FUNCTION_BLOCK SUBL_119_BOTTOM_AND_SIDE_ROUGH_MILLING-SLOT-SIMPLE (* 119-variable local group subscriber *)
  (* Standard: 61499-2 *)
  (* Version 1.0, 10-05-12, GASR, Universidade do Estado de Santa Catarina *)
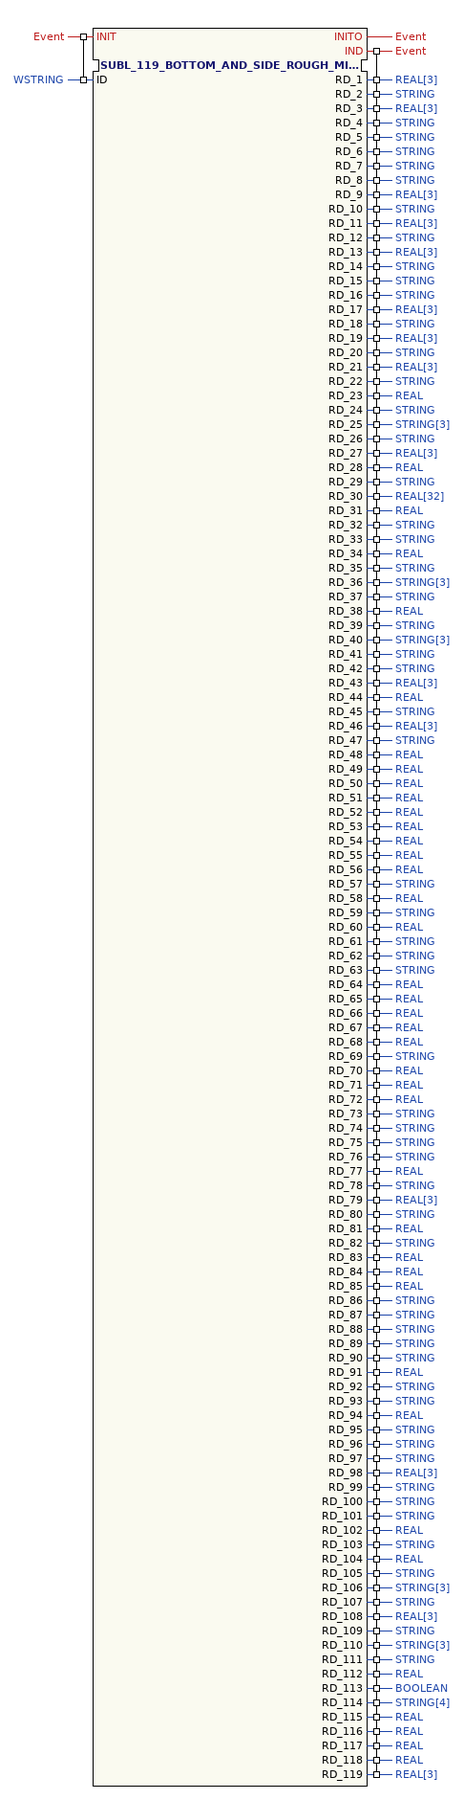
  EVENT_INPUT
    INIT WITH ID; (* Service Initialization *)
  END_EVENT
  EVENT_OUTPUT
    INITO; (* Initialization Confirm *)
    IND WITH RD_1, RD_2, RD_3, RD_4, RD_5, RD_6, RD_7, RD_8, RD_9, RD_10, RD_11, RD_12, RD_13, RD_14, RD_15, RD_16, RD_17, RD_18, RD_19, RD_20, RD_21, RD_22, RD_23, RD_24, RD_25, RD_26, RD_27, RD_28, RD_29, RD_30, RD_31, RD_32, RD_33, RD_34, RD_35, RD_36, RD_37, RD_38, RD_39, RD_40, RD_41, RD_42, RD_43, RD_44, RD_45, RD_46, RD_47, RD_48, RD_49, RD_50, RD_51, RD_52, RD_53, RD_54, RD_55, RD_56, RD_57, RD_58, RD_59, RD_60, RD_61, RD_62, RD_63, RD_64, RD_65, RD_66, RD_67, RD_68, RD_69, RD_70, RD_71, RD_72, RD_73, RD_74, RD_75, RD_76, RD_77, RD_78, RD_79, RD_80, RD_81, RD_82, RD_83, RD_84, RD_85, RD_86, RD_87, RD_88, RD_89, RD_90, RD_91, RD_92, RD_93, RD_94, RD_95, RD_96, RD_97, RD_98, RD_99, RD_100, RD_101, RD_102, RD_103, RD_104, RD_105, RD_106, RD_107, RD_108, RD_109, RD_110, RD_111, RD_112, RD_113, RD_114, RD_115, RD_116, RD_117, RD_118, RD_119; (* Service Indication *)
  END_EVENT
  VAR_INPUT
    ID : WSTRING; (* Default id is the FB instance name *)
  END_VAR
  VAR_OUTPUT
    RD_1 : ARRAY [0..2] OF REAL; (* pos *)
    RD_2 : STRING; (* current_tool *)
    RD_3 : ARRAY [0..2] OF REAL; (* setup.Its_secplane.position.location.coordinates *)
    RD_4 : STRING; (* slot.its_id *)
    RD_5 : STRING; (* its_workpiece.its_id *)
    RD_6 : STRING; (* its_operations.its_id LIST - the list is concatenated in one string *)
    RD_7 : STRING; (* feature_placement.name *)
    RD_8 : STRING; (* feature_placement.location.name *)
    RD_9 : ARRAY [0..2] OF REAL; (* feature_placement.location.coordinates *)
    RD_10 : STRING; (* feature_placement.axis.its_id *)
    RD_11 : ARRAY [0..2] OF REAL; (* feature_placement.axis.direction_ratios *)
    RD_12 : STRING; (* feature_placement.ref_direction.its_id *)
    RD_13 : ARRAY [0..2] OF REAL; (* feature_placement.ref_direction_ratios *)
    RD_14 : STRING; (* depth.name *)
    RD_15 : STRING; (* depth.position.name *)
    RD_16 : STRING; (* depth.position.location.name *)
    RD_17 : ARRAY [0..2] OF REAL; (* depth.position.location.coordinates *)
    RD_18 : STRING; (* depth.position.axis.its_id *)
    RD_19 : ARRAY [0..2] OF REAL; (* depth.position.axis.direction_ratios *)
    RD_20 : STRING; (* depth.position.ref_direction.its_id *)
    RD_21 : ARRAY [0..2] OF REAL; (* depth.position.ref_direction_ratios *)
    RD_22 : STRING; (* course_of_travel *)
    RD_23 : REAL; (* course_of_travel.var1.theoretical_size *)
    RD_24 : STRING; (* course_of_travel.var1.implicit_tolerance *)
    RD_25 : ARRAY [0..2] OF STRING; (* course_of_travel.var1.{vector}, vector = {upper_limit, lower_limit, significant_digits} or {deviation,grade,its_fitting_type} *)
    RD_26 : STRING; (* course_of_travel.direction.its_id *)
    RD_27 : ARRAY [0..2] OF REAL; (* course_of_travel.direction.direction_ratios *)
    RD_28 : REAL; (* course_of_travel.sweep_angle *)
    RD_29 : STRING; (* swept_shape *)
    RD_30 : ARRAY [0..31] OF REAL; (* swept_shape.variable list *)
    RD_31 : REAL; (* swept_shape.profile_length.its_parameter_value *)
    RD_32 : STRING; (* swept_shape.profile_length.its_parameter_unit *)
    RD_33 : STRING; (* end_condition[1] *)
    RD_34 : REAL; (* end_condition[1].var1.theoretical_size *)
    RD_35 : STRING; (* end_condition[1].var1.implicit_tolerance *)
    RD_36 : ARRAY [0..2] OF STRING; (* end_condition[1].var1.{vector}, vector = {upper_limit, lower_limit, significant_digits} or {deviation,grade,its_fitting_type} *)
    RD_37 : STRING; (* end_condition[2] *)
    RD_38 : REAL; (* end_condition[2].var1.theoretical_size *)
    RD_39 : STRING; (* end_condition[2].var1.implicit_tolerance *)
    RD_40 : ARRAY [0..2] OF STRING; (* end_condition[2].var1.{vector}, vector = {upper_limit, lower_limit, significant_digits} or {deviation,grade,its_fitting_type} *)
    RD_41 : STRING; (* bottom_and_side_rough_milling.its_id *)
    RD_42 : STRING; (* its_toolpath.its_list *)
    RD_43 : ARRAY [0..2] OF REAL; (* its_tool_direction *)
    RD_44 : REAL; (* retract_plane *)
    RD_45 : STRING; (* start_point.name *)
    RD_46 : ARRAY [0..2] OF REAL; (* start_point.coordinates *)
    RD_47 : STRING; (* its_tool.its_id *)
    RD_48 : REAL; (* its_tool.its_tool_body.dimension.diameter *)
    RD_49 : REAL; (* its_tool.its_tool_body.dimension.tool_tip_half_angle *)
    RD_50 : REAL; (* its_tool.its_tool_body.dimension.tool_circumference_angle *)
    RD_51 : REAL; (* its_tool.its_tool_body.dimension.cutting_edge_lenght *)
    RD_52 : REAL; (* its_tool.its_tool_body.dimension.edge_radius *)
    RD_53 : REAL; (* its_tool.its_tool_body.dimension.edge_center_vertical *)
    RD_54 : REAL; (* its_tool.its_tool_body.dimension.edge_center_horizontal *)
    RD_55 : REAL; (* its_tool.its_tool_body.number_of_teeth *)
    RD_56 : REAL; (* its_tool.its_tool_body.hand_of_cut *)
    RD_57 : STRING; (* its_tool.its_tool_body.coolant_through *)
    RD_58 : REAL; (* its_tool.its_tool_body.pilot_length *)
    RD_59 : STRING; (* its_tool.its_tool_body.{other_tool_body_parameter} *)
    RD_60 : REAL; (* its_tool.its_cutting_edge.tool_offset_length *)
    RD_61 : STRING; (* its_tool.its_cutting_edge.its_material.standard_identifier *)
    RD_62 : STRING; (* its_tool.its_cutting_edge.its_material.material_identifier *)
    RD_63 : STRING; (* its_tool.its_cutting_edge.its_material.material_property.{list_of_parameters} *)
    RD_64 : REAL; (* its_tool.its_cutting_edge.its_technological_data.cutting_angle *)
    RD_65 : REAL; (* its_tool.its_cutting_edge.its_technological_data.free_angle *)
    RD_66 : REAL; (* its_tool.its_cutting_edge.its_technological_data.aux_angle *)
    RD_67 : REAL; (* its_tool.its_cutting_edge.expected_tool_life *)
    RD_68 : REAL; (* its_tool.its_cutting_edge.its_technology.feedrate *)
    RD_69 : STRING; (* its_tool.its_cutting_edge.its_technology.feedrate_reference *)
    RD_70 : REAL; (* its_tool.its_cutting_edge.its_technology.cutspeed *)
    RD_71 : REAL; (* its_tool.its_cutting_edge.its_technology.spindle *)
    RD_72 : REAL; (* its_tool.its_cutting_edge.its_technology.feedrate_per_tooth *)
    RD_73 : STRING; (* its_tool.its_cutting_edge.its_technology.sincronize_spindle_with_feed *)
    RD_74 : STRING; (* its_tool.its_cutting_edge.its_technology.inhibit_feedrate_override *)
    RD_75 : STRING; (* its_tool.its_cutting_edge.its_technology.inhibit_spindle_override *)
    RD_76 : STRING; (* its_tool.its_cutting_edge.its_technology.its_adaptive_control *)
    RD_77 : REAL; (* its_tool.overall_assembly_length *)
    RD_78 : STRING; (* its_tool.direction_for_spindle_orientation.its_id *)
    RD_79 : ARRAY [0..2] OF REAL; (* its_tool.direction_for_spindle_orientation.direction_ratios *)
    RD_80 : STRING; (* its_tool.tool_holder_diameter_for_spindle_orientation *)
    RD_81 : REAL; (* its_technology.feedrate *)
    RD_82 : STRING; (* its_technology.feedrate_reference *)
    RD_83 : REAL; (* its_technology.cutspeed *)
    RD_84 : REAL; (* its_technology.spindle *)
    RD_85 : REAL; (* its_technology.feedrate_per_tooth *)
    RD_86 : STRING; (* its_technology.sincronize_spindle_with_feed *)
    RD_87 : STRING; (* its_technology.inhibit_feedrate_override *)
    RD_88 : STRING; (* its_technology.inhibit_spindle_override *)
    RD_89 : STRING; (* its_technology.its_adaptive_control *)
    RD_90 : STRING; (* its_machine_functions.coolant *)
    RD_91 : REAL; (* its_machine_functions.coolant_pressure *)
    RD_92 : STRING; (* its_machine_functions.mist *)
    RD_93 : STRING; (* its_machine_functions.through_spindle_coolant *)
    RD_94 : REAL; (* its_machine_functions.through_pressure *)
    RD_95 : STRING; (* its_machine_functions.axis_clamping *)
    RD_96 : STRING; (* its_machine_functions.chip_removal *)
    RD_97 : STRING; (* its_machine_functions.oriented_spindle_stop.its_id *)
    RD_98 : ARRAY [0..2] OF REAL; (* its_machine_functions.oriented_spindle_stop.direction_ratios *)
    RD_99 : STRING; (* its_machine_functions.its_process_model.ini_data_file *)
    RD_100 : STRING; (* its_machine_functions.its_process_model.its_type *)
    RD_101 : STRING; (* its_machine_functions.other_functions *)
    RD_102 : REAL; (* overcut_length *)
    RD_103 : STRING; (* approach.tool_orientation.its_id *)
    RD_104 : REAL; (* approach.tool_orientation.direction_ratios *)
    RD_105 : STRING; (* approach.approach_retract_strategy (name of it) *)
    RD_106 : ARRAY [0..2] OF STRING; (* approach.approach_retract_strategy.list of parameters *)
    RD_107 : STRING; (* retract.tool_orientation.its_id *)
    RD_108 : ARRAY [0..2] OF REAL; (* retract.tool_orientation.direction_ratios *)
    RD_109 : STRING; (* retract.approach_retract_strategy (name of it) *)
    RD_110 : ARRAY [0..2] OF STRING; (* retract.approach_retract_strategy.list of parameters *)
    RD_111 : STRING; (* its_machining_strategy *)
    RD_112 : REAL; (* its_machining_strategy.overlap *)
    RD_113 : BOOLEAN; (* its_machining_strategy.allow_multiple_passes *)
    RD_114 : ARRAY [0..3] OF STRING; (* its_machining_strategy.list of parameters *)
    RD_115 : REAL; (* axial_cutting_depth *)
    RD_116 : REAL; (* radial_cutting_depth *)
    RD_117 : REAL; (* allowance_side *)
    RD_118 : REAL; (* allowance_bottom *)
    RD_119 : ARRAY [0..2] OF REAL; (* slot.course_of_travel.placement.location.coordinates *)
  END_VAR
  SERVICE PUBL_119/SUBL_119 (* Data publication service *)
    SEQUENCE normal_establishment
      PUBL_119.INIT(ID) -> PUBL_119.INITO();
      SUBL_119.INIT(ID) -> SUBL_119.INITO();
    END_SEQUENCE
    SEQUENCE normal_data_transfer
      PUBL_119.REQ(SD_1,SD_2,SD_3,SD_4,SD_5,SD_6,SD_7,SD_8,SD_9,SD_10,SD_11,SD_12,SD_13,SD_14,SD_15,SD_16,SD_17,SD_18,SD_19,SD_20,SD_21,SD_22,SD_23,SD_24,SD_25,SD_26,SD_27,SD_28,SD_29,SD_30,SD_31,SD_32,SD_33,SD_34,SD_35,SD_36,SD_37,SD_38,SD_39,SD_40,SD_41,SD_42,SD_43,SD_44,SD_45,SD_46,SD_47,SD_48,SD_49,SD_50,SD_51,SD_52,SD_53,SD_54,SD_55,SD_56,SD_57,SD_58,SD_59,SD_60,SD_61,SD_62,SD_63,SD_64,SD_65,SD_66,SD_67,SD_68,SD_69,SD_70,SD_71,SD_72,SD_73,SD_74,SD_75,SD_76,SD_77,SD_78,SD_79,SD_80,SD_81,SD_82,SD_83,SD_84,SD_85,SD_86,SD_87,SD_88,SD_89,SD_90,SD_91,SD_92,SD_93,SD_94,SD_95,SD_96,SD_97,SD_98,SD_99,SD_100,SD_101,SD_102,SD_103,SD_104,SD_105,SD_106,SD_107,SD_108,SD_109,SD_110,SD_111,SD_112,SD_113,SD_114,SD_115,SD_116,SD_117,SD_118,SD_119) -> SUBL_119.IND(RD_1,RD_2,RD_3,RD_4,RD_5,RD_6,RD_7,RD_8,RD_9,RD_10,RD_11,RD_12,RD_13,RD_14,RD_15,RD_16,RD_17,RD_18,RD_19,RD_20,RD_21,RD_22,RD_23,RD_24,RD_25,RD_26,RD_27,RD_28,RD_29,RD_30,RD_31,RD_32,RD_33,RD_34,RD_35,RD_36,RD_37,RD_38,RD_39,RD_40,RD_41,RD_42,RD_43,RD_44,RD_45,RD_46,RD_47,RD_48,RD_49,RD_50,RD_51,RD_52,RD_53,RD_54,RD_55,RD_56,RD_57,RD_58,RD_59,RD_60,RD_61,RD_62,RD_63,RD_64,RD_65,RD_66,RD_67,RD_68,RD_69,RD_70,RD_71,RD_72,RD_73,RD_74,RD_75,RD_76,RD_77,RD_78,RD_79,RD_80,RD_81,RD_82,RD_83,RD_84,RD_85,RD_86,RD_87,RD_88,RD_89,RD_90,RD_91,RD_92,RD_93,RD_94,RD_95,RD_96,RD_97,RD_98,RD_99,RD_100,RD_101,RD_102,RD_103,RD_104,RD_105,RD_106,RD_107,RD_108,RD_109,RD_110,RD_111,RD_112,RD_113,RD_114,RD_115,RD_116,RD_117,RD_118,RD_119);
    END_SEQUENCE
  END_SERVICE
END_FUNCTION_BLOCK
